Omron CX-Programmer project NewProject (CX-Programmer 9.73)

# PLC NewPLC1: CP1H XA

## Global symbols (name address type ; comment)
0.00 BOOL  ; START
0.01 BOOL  ; STOP
0.02 BOOL  ; EMERGENCY
100.00 BOOL  ; HIJAU1
100.01 BOOL  ; KUNING1
100.02 BOOL  ; MERAH1
100.03 BOOL  ; HIJAU2
100.04 BOOL  ; KUNING2
100.05 BOOL  ; MERAH2
100.06 BOOL  ; HIJAU3
100.07 BOOL  ; KUNING3
100.08 BOOL  ; MERAH3
100.09 BOOL  ; HIJAU4
100.10 BOOL  ; KUNING4
100.11 BOOL  ; MERAH4
100.12 BOOL  ; NO_RIGHT_TURN
100.13 BOOL  ; DONT_GO_THIS_WAY
101.00 BOOL  ; WARNING
A352 CHANNEL  ; JAM TANGGAL
A354 CHANNEL  ; HARI
D0.00 BOOL  ; t008
D100 CHANNEL  ; DETIK
D101 CHANNEL  ; MENIT
D102 CHANNEL  ; JAM
D103 CHANNEL  ; HARI
W0.00 BOOL  ; HOLD
W0.01 BOOL  ; MAIN
W0.02 BOOL  ; KONDISI1
W0.03 BOOL  ; KONDISI2
W0.04 BOOL  ; DUMMY

## Program NewProgram1 (cyclic task 0)
Local symbols
MERAH3 BOOL

### Section Section1

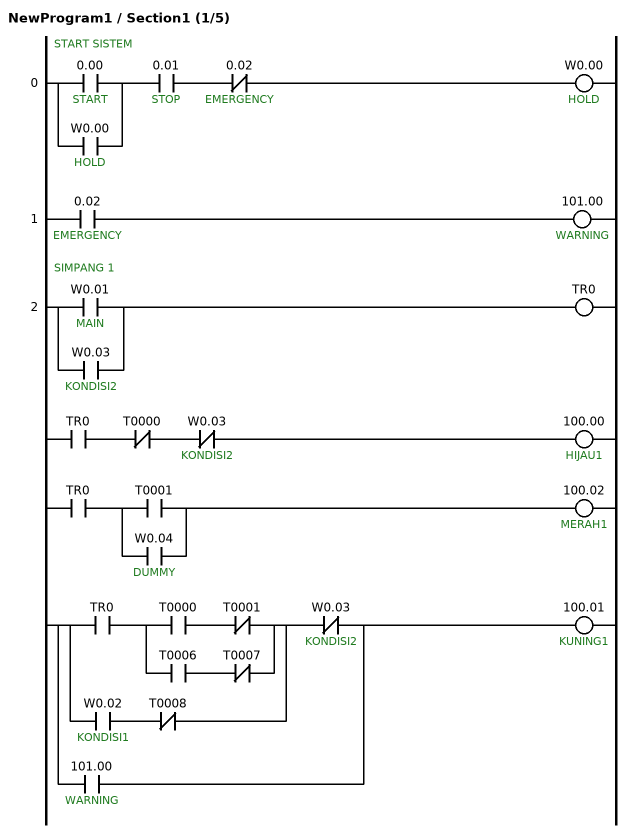
; rung 0: START SISTEM
LD 0.00  ; START
OR W0.00  ; HOLD
AND 0.01  ; STOP
ANDNOT 0.02  ; EMERGENCY
OUT W0.00  ; HOLD
; rung 1
LD 0.02  ; EMERGENCY
OUT 101.00  ; WARNING
; rung 2: SIMPANG 1
LD W0.01  ; MAIN
OR W0.03  ; KONDISI2
OUT TR0
ANDNOT T0000
ANDNOT W0.03  ; KONDISI2
OUT 100.00  ; HIJAU1
LD TR0
LD T0001
OR W0.04  ; DUMMY
ANDLD
OUT 100.02  ; MERAH1
LD TR0
LD T0000
ANDNOT T0001
LD T0006
ANDNOT T0007
ORLD
ANDLD
LD W0.02  ; KONDISI1
ANDNOT T0008
ORLD
ANDNOT W0.03  ; KONDISI2
OR 101.00  ; WARNING
OUT 100.01  ; KUNING1

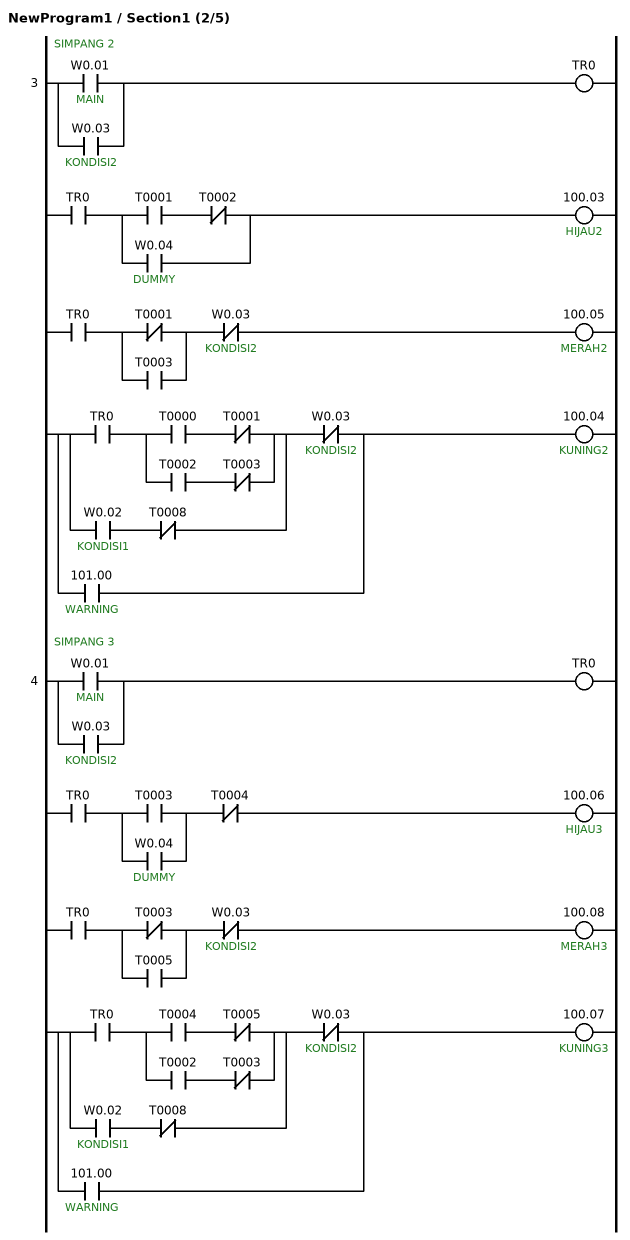
; rung 3: SIMPANG 2
LD W0.01  ; MAIN
OR W0.03  ; KONDISI2
OUT TR0
LD T0001
ANDNOT T0002
OR W0.04  ; DUMMY
ANDLD
OUT 100.03  ; HIJAU2
LD TR0
LDNOT T0001
OR T0003
ANDLD
ANDNOT W0.03  ; KONDISI2
OUT 100.05  ; MERAH2
LD TR0
LD T0000
ANDNOT T0001
LD T0002
ANDNOT T0003
ORLD
ANDLD
LD W0.02  ; KONDISI1
ANDNOT T0008
ORLD
ANDNOT W0.03  ; KONDISI2
OR 101.00  ; WARNING
OUT 100.04  ; KUNING2
; rung 4: SIMPANG 3
LD W0.01  ; MAIN
OR W0.03  ; KONDISI2
OUT TR0
LD T0003
OR W0.04  ; DUMMY
ANDLD
ANDNOT T0004
OUT 100.06  ; HIJAU3
LD TR0
LDNOT T0003
OR T0005
ANDLD
ANDNOT W0.03  ; KONDISI2
OUT 100.08  ; MERAH3
LD TR0
LD T0004
ANDNOT T0005
LD T0002
ANDNOT T0003
ORLD
ANDLD
LD W0.02  ; KONDISI1
ANDNOT T0008
ORLD
ANDNOT W0.03  ; KONDISI2
OR 101.00  ; WARNING
OUT 100.07  ; KUNING3

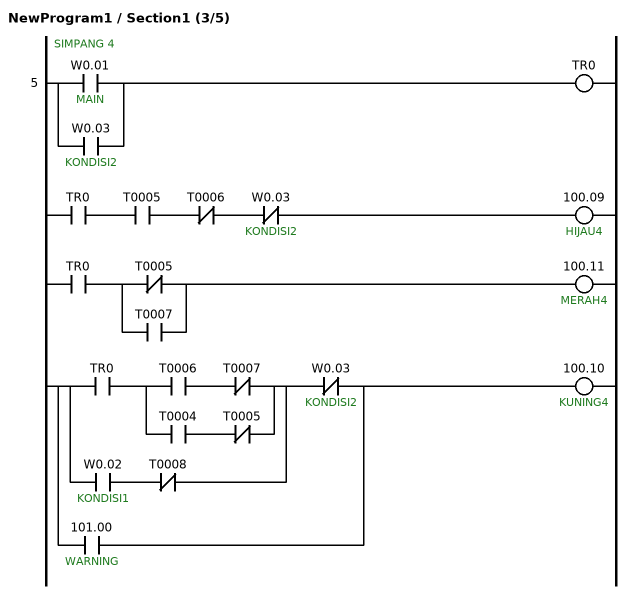
; rung 5: SIMPANG 4
LD W0.01  ; MAIN
OR W0.03  ; KONDISI2
OUT TR0
AND T0005
ANDNOT T0006
ANDNOT W0.03  ; KONDISI2
OUT 100.09  ; HIJAU4
LD TR0
LDNOT T0005
OR T0007
ANDLD
OUT 100.11  ; MERAH4
LD TR0
LD T0006
ANDNOT T0007
LD T0004
ANDNOT T0005
ORLD
ANDLD
LD W0.02  ; KONDISI1
ANDNOT T0008
ORLD
ANDNOT W0.03  ; KONDISI2
OR 101.00  ; WARNING
OUT 100.10  ; KUNING4

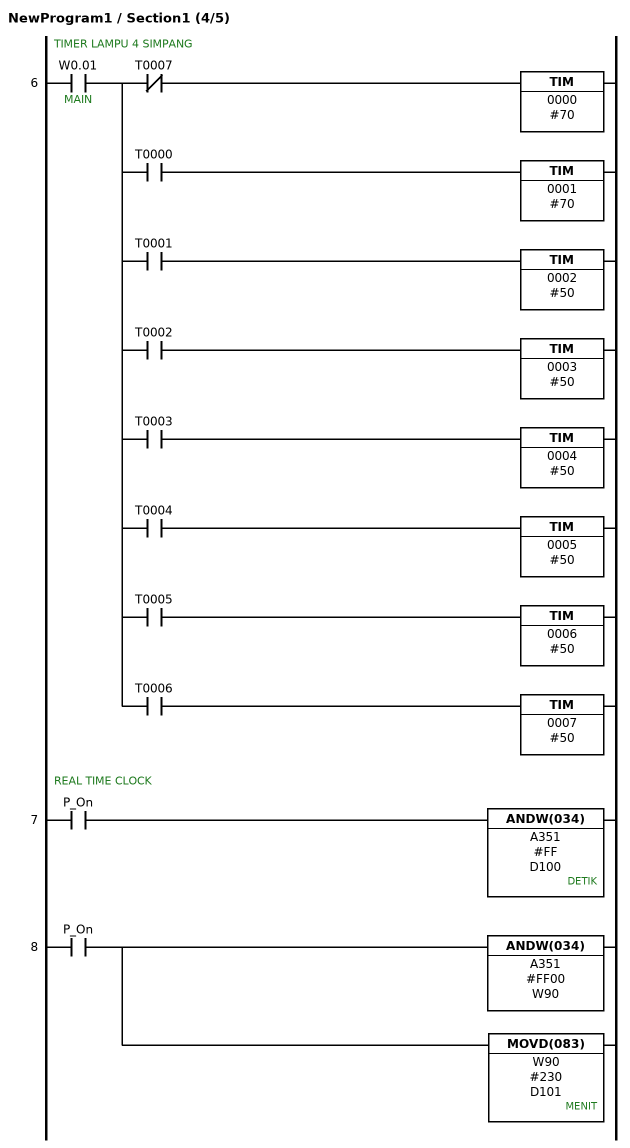
; rung 6: TIMER LAMPU 4 SIMPANG
LD W0.01  ; MAIN
OUT TR0
ANDNOT T0007
TIM 0000 #70
LD TR0
AND T0000
TIM 0001 #70
LD TR0
AND T0001
TIM 0002 #50
LD TR0
AND T0002
TIM 0003 #50
LD TR0
AND T0003
TIM 0004 #50
LD TR0
AND T0004
TIM 0005 #50
LD TR0
AND T0005
TIM 0006 #50
LD TR0
AND T0006
TIM 0007 #50
; rung 7: REAL TIME CLOCK
LD P_On
ANDW(034) A351 #FF D100  ; DETIK
; rung 8
LD P_On
ANDW(034) A351 #FF00 W90
MOVD(083) W90 #230 D101  ; MENIT

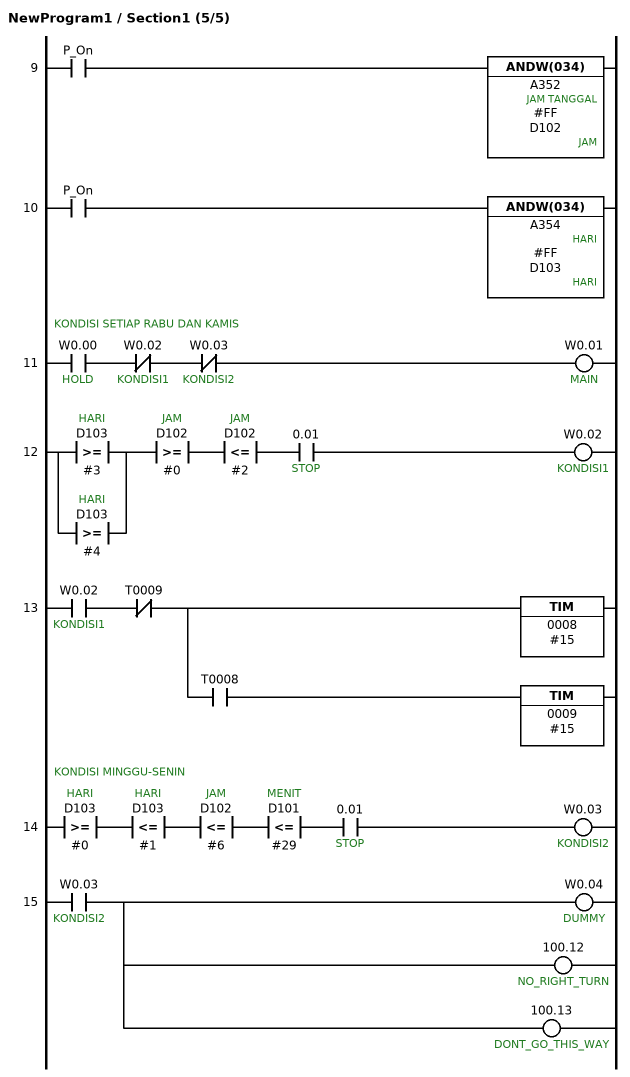
; rung 9
LD P_On
ANDW(034) A352 #FF D102  ; JAM TANGGAL, JAM
; rung 10
LD P_On
ANDW(034) A354 #FF D103  ; HARI
; rung 11: KONDISI SETIAP RABU DAN KAMIS
LD W0.00  ; HOLD
ANDNOT W0.02  ; KONDISI1
ANDNOT W0.03  ; KONDISI2
OUT W0.01  ; MAIN
; rung 12
LD>=(325) D103 #3  ; HARI
OR>=(325) D103 #4  ; HARI
AND>=(325) D102 #0  ; JAM
AND<=(315) D102 #2  ; JAM
AND 0.01  ; STOP
OUT W0.02  ; KONDISI1
; rung 13
LD W0.02  ; KONDISI1
ANDNOT T0009
TIM 0008 #15
AND T0008
TIM 0009 #15
; rung 14: KONDISI MINGGU-SENIN
LD>=(325) D103 #0  ; HARI
AND<=(315) D103 #1  ; HARI
AND<=(315) D102 #6  ; JAM
AND<=(315) D101 #29  ; MENIT
AND 0.01  ; STOP
OUT W0.03  ; KONDISI2
; rung 15
LD W0.03  ; KONDISI2
OUT W0.04  ; DUMMY
OUT 100.12  ; NO_RIGHT_TURN
OUT 100.13  ; DONT_GO_THIS_WAY

### Section END
; rung 0
END(001)